// TIA Portal V20 export
DATA_BLOCK "BlowOffValve_DB"   // DB550
// stored: AutoNumber false, InstanceOfName BlowOffValve, InstanceOfType FB
"BlowOffValve"
   // VAR
   //    Var { ExternalAccessible := 'False'; ExternalVisible := 'False'; ExternalWritable := 'False'} : "TypeVar";
   //    T { ExternalAccessible := 'False'; ExternalVisible := 'False'; ExternalWritable := 'False'} : Array[1..20] of IEC_TIMER;
   //    blowOff { ExternalAccessible := 'False'; ExternalVisible := 'False'; ExternalWritable := 'False'} : Bool;
   //    breakTime { ExternalAccessible := 'False'; ExternalVisible := 'False'; ExternalWritable := 'False'} : Time;
   //    intervallTime { ExternalAccessible := 'False'; ExternalVisible := 'False'; ExternalWritable := 'False'} : Time;
   //    intervallTimeOff { ExternalAccessible := 'False'; ExternalVisible := 'False'; ExternalWritable := 'False'} : Time;
   //    bottom { ExternalAccessible := 'False'; ExternalVisible := 'False'; ExternalWritable := 'False'} : Struct
   //       delayStart : Time;
   //       Impuls : Time;
   //       start : Bool;
   //       blowOff : Bool;
   //    END_STRUCT;
   //    left { ExternalAccessible := 'False'; ExternalVisible := 'False'; ExternalWritable := 'False'} : Struct
   //       delayStart : Time;
   //       Impuls : Time;
   //       start : Bool;
   //       blowOff : Bool;
   //    END_STRUCT;
   //    right { ExternalAccessible := 'False'; ExternalVisible := 'False'; ExternalWritable := 'False'} : Struct
   //       delayStart : Time;
   //       Impuls : Time;
   //       start : Bool;
   //       blowOff : Bool;
   //    END_STRUCT;
   //    xray { ExternalAccessible := 'False'; ExternalVisible := 'False'; ExternalWritable := 'False'} : Struct
   //       delayStart : Time;
   //       Impuls : Time;
   //       start : Bool;
   //       blowOff : Bool;
   //    END_STRUCT;
   // END_VAR
BEGIN
END_DATA_BLOCK
